FUNCTION_BLOCK AutoState IMPLEMENTS I_SD_ValveState
VAR_INPUT
END_VAR
VAR_OUTPUT
END_VAR
VAR
    _ptSdValve : POINTER TO SD_Valve;
END_VAR

METHOD Close : BOOL
Close := TRUE;
END_METHOD

METHOD FB_init : BOOL
VAR_INPUT
	bInitRetains : BOOL; // if TRUE, the retain variables are initialized (warm start / cold start)
	bInCopyCode : BOOL;  // if TRUE, the instance afterwards gets moved into the copy code (online change)
    ptSdValve : POINTER TO SD_Valve;
END_VAR
_ptSdValve := ptSdValve;
END_METHOD

METHOD Open : BOOL
Open := true;
END_METHOD

METHOD RUN
THIS^();
END_METHOD

PROPERTY StateName : STRING
GET
StateName := 'Auto';
END_GET
END_PROPERTY

END_FUNCTION_BLOCK

(* stored: Version 1.1.0.1, ProductVersion 3.1.4024.12
   POU AutoState: Id {8cea08e5-a635-4ec2-8d51-b4eb2b4b528e}, SpecialFunc None
   Method Close: Id {32e551a6-420e-4bc8-be73-27bc5964241a}
   Method FB_init: Id {1fdcbc93-77bb-49d9-b6de-6b6192030d9d}
   Method Open: Id {0ee2d403-d4f1-4413-92cc-9dccb688ee67}
   Method RUN: Id {41fec5c8-d503-4e81-91ea-83fd3de9434b}
   Property StateName: Id {b579d6c8-3340-4fe9-95b6-8f4102fdbb32}
   Get Get: Id {a9de4539-3d12-48ce-bd37-3fa7eed1aad3} *)
